// Block: Encoder

DATA_BLOCK Encoder
{ S7_Optimized_Access := 'TRUE' }
VERSION : 0.1
   NON_RETAIN
   VAR
      "1248A1" : PD_TEL81;
   END_VAR

BEGIN
   // No initialization required
END_DATA_BLOCK
